//---------------------------------------------------------------------------------------------------------------
//
//  HAUD 2023.12.19
//
//  - XTS_TRANSPORT_LAYER
//
//  fb_Mover
//  - all positioning input is modulo value
//  - wrap MC function blocks
//
//
//---------------------------------------------------------------------------------------------------------------
// This SOFTWARE is provided as an Example by THE PROVIDER "as is" and "with all faults." THE PROVIDER makes no 
// representations or warranties of any kind concerning the safety, suitability, lack of viruses, inaccuracies, 
// typographical errors, or other harmful components of this SOFTWARE. There are inherent dangers in the use of 
// any software, and you are solely responsible for determining whether this SOFTWARE is compatible with your 
// equipment and other software installed on your equipment. You are also solely responsible for the protection 
// of your equipment and backup of your data, and THE PROVIDER will not be liable for any damages you may suffer 
// in connection with using, modifying, or distributing this SOFTWARE.
//---------------------------------------------------------------------------------------------------------------
FUNCTION_BLOCK fb_Mover IMPLEMENTS I_XtsTransport_Mover
VAR
  _nMoverId         : UINT;

  _sState           : STRING;

  _Master,
  _Mover            : REFERENCE TO AXIS_REF;
  _rLastPosition    : REFERENCE TO LREAL;
  _rLastGap         : REFERENCE TO LREAL;

  _RailLength       : LREAL;
  _nSyncStrategy    : Tc3_Mc3Definitions.MC_SYNC_STRATEGY := Tc3_Mc3Definitions.MC_SYNC_STRATEGY.mcSyncStrategySlow; // minimal movement with this strategy 

  // mover compact axis information
  _stInfo           : REFERENCE TO ST_MOVER_INFO; // ActPos, Enable, ...

  _bError           : BOOL;   // used in Cycle()
  _nErrorIdMover,             // used in Cycle()
  _nErrorIdPower    : UDINT;  // used in Cycle()

  //---------------------------------------------------------------------------
  // MC2 and CA function blocks
  //---------------------------------------------------------------------------
  _wMoverState      : DWORD;

  _fbMoveAbsCa      : Tc3_McCollisionAvoidance.MC_MoveAbsoluteCA;
  _fbSendAbsCa      : Tc3_McCollisionAvoidance.MC_MoveAbsoluteCA;
  _fbGearInPosCa    : Tc3_McCollisionAvoidance.MC_GearInPosCA;
  _fbHaltCa         : Tc3_McCollisionAvoidance.MC_HaltCA;

  _fbMoveAbs        : Tc2_MC2.MC_MoveAbsolute;
  _fbHalt           : Tc2_MC2.MC_Halt;
  _fbReset          : Tc2_MC2.MC_Reset;
  _fbStop           : Tc2_MC2.MC_Stop;

  _fbGearIn         : Tc2_MC2.MC_GearIn;
  _fbGearOut        : Tc2_MC2.MC_GearOut;

  _fbPower          : Tc2_MC2.MC_Power;

  _stMsg            : ST_Message;
  _eMessageLevel    : E_MessageType;
END_VAR

METHOD Check : BOOL
// check The thing that should not be

IF NOT (_nMoverId > 0)
THEN
  _sState                     := 'Mover: missing ID';
  RETURN;
END_IF

IF NOT __ISVALIDREF(_Mover)
THEN
  _sState                     := 'Mover: missing pointer';
  RETURN;
END_IF

IF NOT __ISVALIDREF(_rLastPosition)
THEN
  _sState                     := '_rLastPosition: missing pointer';
  RETURN;
END_IF

IF NOT __ISVALIDREF(_rLastGap)
THEN
  _sState                     := '_rLastGap: missing pointer';
  RETURN;
END_IF

IF NOT __ISVALIDREF(_stInfo)
THEN
  _sState                     := '_stInfo: missing pointer';
  RETURN;
END_IF

_sState                       := 'CHECK_DONE';
Check                         := TRUE;
END_METHOD

METHOD Cycle : E_PROGRESS
VAR_INST
  _eState             : E_PROGRESS;

  _rtrigMoverError,
  _rtrigPowerError    : Tc2_Standard.R_TRIG;
END_VAR
IF NOT Check() THEN Cycle := E_PROGRESS.PROGRESS_ERROR; RETURN; END_IF

_stMsg.eDevice            := e_Device.Mover + _nMoverId;

//-----------------------------------------------------------------------------------------------
// cyclic NC mapping
//-----------------------------------------------------------------------------------------------
_Mover();
//-----------------------------------------------------------------------------------------------


//-----------------------------------------------------------------------------------------------
// cyclic MC_Power
//-----------------------------------------------------------------------------------------------
_fbPower(
        Axis              := _Mover, 
        Enable_Positive   := TRUE, 
        Enable_Negative   := TRUE, 
        BufferMode        := MC_BufferMode.MC_Aborting);

_rtrigPowerError(CLK := _fbPower.Error);
_rtrigMoverError(CLK := _Mover.Status.Error); 

IF _rtrigMoverError.Q
THEN
  _bError                 := TRUE;  // deleted by Reset()
  // catch error
  _nErrorIdMover          := _Mover.Status.ErrorID;
  _stInfo.nErrorId        := _nErrorIdMover;

  _stMsg.eType            := E_MessageType.eMessageError;
  _stMsg.eSubdevice       := e_Subdevice.AxisControl;
  _stMsg.iErrorNumber     := _nErrorIdMover;
  _stMsg.sText            := 'Axis Error';
  f_MessageSet(_stMsg);
END_IF

IF _rtrigPowerError.Q
THEN
  _bError                 := TRUE;  // deleted by Reset()
  // catch error
  _nErrorIdPower          := _fbPower.ErrorID;
  _stInfo.nErrorId        := _nErrorIdPower;

  _stMsg.eType            := E_MessageType.eMessageError;
  _stMsg.eSubdevice       := e_Subdevice.AxisControl;
  _stMsg.iErrorNumber     := _nErrorIdMover;
  _stMsg.sText            := 'Axis Error';
  f_MessageSet(_stMsg);
END_IF
//-----------------------------------------------------------------------------------------------

//-----------------------------------------------------------------------------------------------
// cyclic state
//-----------------------------------------------------------------------------------------------
IF NOT _Mover.Status.ControlLoopClosed
THEN
  _eState                       := E_PROGRESS.PROGRESS_INIT;
ELSE
  _eState                       := E_PROGRESS.PROGRESS_WORKING;
END_IF
 
IF _bError
THEN
  _eState                       := E_PROGRESS.PROGRESS_ERROR;
END_IF
//-----------------------------------------------------------------------------------------------


//-----------------------------------------------------------------------------
// cyclic Mover info data
// get collision avoiding information from cyclic interface
//-----------------------------------------------------------------------------------------------
memcpy(ADR(_wMoverState), ADR(_Mover.NcToPlc.StateDWord2), SIZEOF(_wMoverState));

_stInfo.bMoverEnabled           := _Mover.Status.ControlLoopClosed;
_stInfo.bMoverError             := _bError;
_stInfo.bMoverCoupled           := _Mover.Status.Coupled;
_stInfo.bMoverStandstill        := _Mover.Status.NotMoving;
_stInfo.bMoverAvoidingCollision := _wMoverState.0;

_stInfo.rModuloActPos           := TO_REAL(_Mover.NcToPlc.ModuloActPos);
_stInfo.rAbsActPos              := TO_REAL(_Mover.NcToPlc.ActPos);

_stInfo.rModuloTargetPos        := TO_REAL(Tc2_Math.LMOD(_rLastPosition, _RailLength));
_stInfo.rAbsTargetPos           := TO_REAL(_rLastPosition);

IF (_Mover.NcToPlc.ActPos < _rLastPosition + 0.05) AND
   (_Mover.NcToPlc.ActPos > _rLastPosition - 0.05)
THEN
  _stInfo.bMoverInTarget        := TRUE;
ELSE
  _stInfo.bMoverInTarget        := FALSE;
END_IF
//-----------------------------------------------------------------------------

Cycle                           := _eState;
END_METHOD

METHOD Disable : E_PROGRESS
VAR_INPUT
  Execute             : BOOL;
END_VAR
VAR_INST
  _nErrorId           : UDINT;
  _eState             : E_PROGRESS;
END_VAR
IF NOT Execute THEN _eState  := E_PROGRESS.PROGRESS_INIT; END_IF 
IF NOT Check() THEN Disable  := E_PROGRESS.PROGRESS_ERROR; RETURN; END_IF


CASE _eState
OF
  E_PROGRESS.PROGRESS_INIT:
    IF Execute
    THEN
      _nErrorId               := 0;
      _eState                 := E_PROGRESS.PROGRESS_BUSY;
    END_IF
END_CASE
//-----------------------------------------------------------------------------
//-----------------------------------------------------------------------------
CASE _eState
OF
  E_PROGRESS.PROGRESS_BUSY:
    _eState                   := E_PROGRESS.PROGRESS_PREPARE;
    _fbPower.Enable           := FALSE;
END_CASE
//-----------------------------------------------------------------------------
//-----------------------------------------------------------------------------
CASE _eState
OF
  E_PROGRESS.PROGRESS_PREPARE:
    IF (_fbPower.Error)
    THEN
      _eState                 := E_PROGRESS.PROGRESS_ERROR;
      _nErrorId               := _fbPower.ErrorId;

      _stMsg.eType            := E_MessageType.eMessageError;
      _stMsg.eSubdevice       := e_Subdevice.fbPower;
      _stMsg.iErrorNumber     := _nErrorId;
      _stMsg.sText            := concat('Axis Disable: ', TO_STRING(_eState));
      f_MessageSet(_stMsg);

    ELSIF NOT (_Mover.Status.ControlLoopClosed)
    THEN
      _eState                 := E_PROGRESS.PROGRESS_DONE;

      IF (_eMessageLevel > E_MessageType.eMessageError)
      THEN
        _stMsg.eType          := E_MessageType.eMessageInfo;
        _stMsg.eSubdevice     := e_Subdevice.fbPower;
        _stMsg.iErrorNumber   := 0;
        _stMsg.sText          := concat('Axis Disable: ', TO_STRING(_eState));
        f_MessageSet(_stMsg);
      END_IF
    END_IF
END_CASE
//-----------------------------------------------------------------------------
//-----------------------------------------------------------------------------

Disable                       := _eState;
END_METHOD

METHOD Enable : E_PROGRESS
VAR_INPUT
  Execute             : BOOL;
END_VAR
VAR_INST
  _nErrorId           : UDINT;
  _eState             : E_PROGRESS;
END_VAR
IF NOT Execute THEN _eState  := E_PROGRESS.PROGRESS_INIT; END_IF 
IF NOT Check() THEN Enable   := E_PROGRESS.PROGRESS_ERROR; RETURN; END_IF


CASE _eState
OF
  E_PROGRESS.PROGRESS_INIT:
    IF Execute
    THEN
      _nErrorId               := 0;
      _eState                 := E_PROGRESS.PROGRESS_BUSY;
    END_IF
END_CASE
//-----------------------------------------------------------------------------
//-----------------------------------------------------------------------------
CASE _eState
OF
  E_PROGRESS.PROGRESS_BUSY:
    _eState                   := E_PROGRESS.PROGRESS_PREPARE;
    _fbPower.Enable           := TRUE;
END_CASE
//-----------------------------------------------------------------------------
//-----------------------------------------------------------------------------
CASE _eState
OF
  E_PROGRESS.PROGRESS_PREPARE:
    IF (_fbPower.Error)
    THEN
      _eState                 := E_PROGRESS.PROGRESS_ERROR;
      _nErrorId               := _fbPower.ErrorId;
      _stInfo.nErrorId        := _nErrorId;

      _stMsg.eType            := E_MessageType.eMessageError;
      _stMsg.eSubdevice       := e_Subdevice.fbPower;
      _stMsg.iErrorNumber     := _nErrorId;
      _stMsg.sText            := concat('Axis Enable: ', TO_STRING(_eState));
      f_MessageSet(_stMsg);

    ELSIF (_Mover.Status.ControlLoopClosed)
    THEN
      _eState                 := E_PROGRESS.PROGRESS_DONE;

      IF (_eMessageLevel > E_MessageType.eMessageError)
      THEN
        _stMsg.eType          := E_MessageType.eMessageInfo;
        _stMsg.eSubdevice     := e_Subdevice.fbPower;
        _stMsg.iErrorNumber   := _nErrorId;
        _stMsg.sText          := concat('Axis Enable: ', TO_STRING(_eState));
        f_MessageSet(_stMsg);
      END_IF
    END_IF
END_CASE
//-----------------------------------------------------------------------------
//-----------------------------------------------------------------------------

Enable                   := _eState;
END_METHOD

METHOD GearIn : E_PROGRESS;
VAR_INPUT
  Execute             : BOOL;
  stMoveData          : ST_MOVE_DATA;
  stGearData          : ST_GEAR_DATA;
END_VAR
VAR_INST
  _nErrorId           : UDINT;
  _eState             : E_PROGRESS;
END_VAR
IF NOT Execute THEN _eState  := E_PROGRESS.PROGRESS_INIT; END_IF 
IF NOT Check() THEN GearIn   := E_PROGRESS.PROGRESS_ERROR; RETURN; END_IF


CASE _eState
OF
  E_PROGRESS.PROGRESS_INIT:
    IF Execute
    THEN
      _nErrorId               := 0;
      _eState                 := E_PROGRESS.PROGRESS_BUSY;

      IF NOT __ISVALIDREF(_Master)
      THEN
        _bError               := TRUE;
        _nErrorId             := 666;
        _eState               := E_PROGRESS.PROGRESS_ERROR;

        _stMsg.eType          := E_MessageType.eMessageError;
        _stMsg.eSubdevice     := e_Subdevice.fbGearIn;
        _stMsg.iErrorNumber   := _nErrorId;
        _stMsg.sText          := concat('Invalid Master Ref: ', TO_STRING(_eState));
        f_MessageSet(_stMsg);
      END_IF
    END_IF
END_CASE
//-----------------------------------------------------------------------------
//-----------------------------------------------------------------------------
CASE _eState
OF
  E_PROGRESS.PROGRESS_BUSY:
    _eState                   := E_PROGRESS.PROGRESS_PREPARE;
    _fbPower.Override         := stMoveData.rOverride;

    _fbGearIn(
            Master            := _Master, 
            Slave             := _Mover,
            Execute           := FALSE,
            RatioNumerator    := stGearData.rGearNumerator,
            RatioDenominator  := stGearData.iGearDenumerator, 
            Acceleration      := stMoveData.rAcc, 
            Deceleration      := stMoveData.rAcc, 
            Jerk              := stMoveData.rJerk, 
            BufferMode        := Tc2_MC2.MC_BufferMode.MC_Aborting);
END_CASE
//-----------------------------------------------------------------------------
//-----------------------------------------------------------------------------
CASE _eState
OF
  E_PROGRESS.PROGRESS_PREPARE:
    _fbGearIn(
            Master            := _Master, 
            Slave             := _Mover,
            Execute           := TRUE);

    IF _fbGearIn.Error
    THEN
      _bError                 := TRUE;
      _nErrorId               := _fbGearIn.ErrorID;
      _eState                 := E_PROGRESS.PROGRESS_ERROR;

      _stMsg.eType            := E_MessageType.eMessageError;
      _stMsg.eSubdevice       := e_Subdevice.fbGearIn;
      _stMsg.iErrorNumber     := _nErrorId;
      _stMsg.sText            := TO_STRING(_eState);
      f_MessageSet(_stMsg);

    ELSIF _fbGearIn.InGear
    THEN
      _eState                 := E_PROGRESS.PROGRESS_DONE;

      IF (_eMessageLevel > E_MessageType.eMessageError)
      THEN
        _stMsg.eType          := E_MessageType.eMessageInfo;
        _stMsg.eSubdevice     := e_Subdevice.fbGearIn;
        _stMsg.iErrorNumber   := _nErrorId;
        _stMsg.sText          := TO_STRING(_eState);
        f_MessageSet(_stMsg);
      END_IF
    END_IF
END_CASE
//-----------------------------------------------------------------------------
//-----------------------------------------------------------------------------
CASE _eState
OF
  E_PROGRESS.PROGRESS_ERROR,
  E_PROGRESS.PROGRESS_DONE:
    _stInfo.nErrorId          := _nErrorId;
    _fbGearIn(
            Master            := _Master, 
            Slave             := _Mover,
            Execute           := FALSE);
END_CASE
//-----------------------------------------------------------------------------
//-----------------------------------------------------------------------------

GearIn                        := _eState;
END_METHOD

METHOD GearInPosCa : E_PROGRESS
VAR_INPUT
  Execute             : BOOL;
  stMoveData          : ST_MOVE_DATA;
  stGearData          : ST_GEAR_DATA;  
END_VAR
VAR_INST
  _nErrorId           : UDINT;
  _rPosLate,
  _rPos               : LREAL;
  _eState             : E_PROGRESS;

  _rModActPos         : LREAL;
END_VAR
IF NOT Execute THEN _eState       := E_PROGRESS.PROGRESS_INIT; END_IF 
IF NOT Check() THEN GearInPosCa   := E_PROGRESS.PROGRESS_ERROR; RETURN; END_IF


CASE _eState
OF
  E_PROGRESS.PROGRESS_INIT:
    IF Execute
    THEN
      _rPosLate               := 0.0;
      _nErrorId               := 0;
      _eState                 := E_PROGRESS.PROGRESS_BUSY;
      _rModActPos             := Tc2_Math.LMOD(_Mover.NcToPlc.SetPos, _RailLength);

      IF NOT __ISVALIDREF(_Master)
      THEN
        _bError               := TRUE;
        _nErrorId             := 666;
        _eState               := E_PROGRESS.PROGRESS_ERROR;

        _stMsg.eType          := E_MessageType.eMessageError;
        _stMsg.eSubdevice     := e_Subdevice.fbGearInPosCa;
        _stMsg.iErrorNumber   := _nErrorId;
        _stMsg.sText          := concat('Invalid Master Ref: ', TO_STRING(_eState));
        f_MessageSet(_stMsg);

      ELSIF (_rModActPos > stGearData.rModuloSyncPosSlave + stMoveData.rDelta)
      THEN
        _bError               := TRUE;
        _rPosLate             := _rModActPos;
        _rPos                 := stGearData.rModuloSyncPosSlave + stMoveData.rDelta;

        _nErrorId             := 667;
        _eState               := E_PROGRESS.PROGRESS_ERROR;

        _stMsg.eType          := E_MessageType.eMessageError;
        _stMsg.eSubdevice     := e_Subdevice.fbGearInPosCa;
        _stMsg.iErrorNumber   := _nErrorId;
        _stMsg.sText          := concat('_rModActPos: ', TO_STRING(_rPosLate));
        _stMsg.sText          := concat(_stMsg.sText, '; ModuloSyncPosSlave + stMoveData.Delta: ');
        _stMsg.sText          := concat(_stMsg.sText, TO_STRING(_rPos));
        f_MessageSet(_stMsg);
      END_IF
    END_IF
END_CASE
//-----------------------------------------------------------------------------
//-----------------------------------------------------------------------------
CASE _eState
OF
  E_PROGRESS.PROGRESS_BUSY:
    _eState                   := E_PROGRESS.PROGRESS_PREPARE;

    _fbPower.Override         := stMoveData.rOverride;

    _fbGearInPosCa(
        Master                := _Master, 
        Slave                 := _Mover, 
        Execute               := FALSE, 
        ContinuousUpdate      := TRUE, 
        RatioNumerator        := stGearData.rGearNumerator, 
        RatioDenumerator      := stGearData.iGearDenumerator, 

        MasterSyncPosition    := _Master.NcToPlc.ActPos 
                               + stGearData.rDeltaToMasterPos,                            // absolute position

        SlaveSyncPosition     := ABS(_Mover.NcToPlc.ModuloActTurns)*_RailLength
                               + stGearData.rModuloSyncPosSlave,                          // absolute position

        SyncStrategy          := _nSyncStrategy,  
        SyncMode              := Tc3_Mc3Definitions.MC_SYNC_MODE.mcSyncModeNonModulo,     // all positions as absolute value
        MasterStartDistance   := stGearData.rMasterStartDistance,                         // if <> 0 --> master has to move before this fb does anything
        Velocity              := stMoveData.rVelo, 
        Acceleration          := stMoveData.rAcc, 
        Deceleration          := stMoveData.rAcc, 
        Jerk                  := stMoveData.rJerk, 
        Gap                   := stMoveData.rGap, 
        BufferMode            := Tc3_Mc3Definitions.MC_BUFFER_MODE.mcAborting);

        IF (_eMessageLevel > E_MessageType.eMessageInfo)
        THEN
          _stMsg.eType        := E_MessageType.eMessageVerbose;
          _stMsg.eSubdevice   := e_Subdevice.fbGearInPosCa;
          _stMsg.iErrorNumber := _nErrorId;
          _stMsg.sText        := TO_STRING(_eState);
          f_MessageSet(_stMsg);
        END_IF
END_CASE
//-----------------------------------------------------------------------------
//-----------------------------------------------------------------------------
CASE _eState
OF
  E_PROGRESS.PROGRESS_PREPARE:
    _fbGearInPosCa(
        Master                := _Master, 
        Slave                 := _Mover, 
        Execute               := TRUE, 
        ContinuousUpdate      := TRUE);

    IF _fbGearInPosCa.Error
    THEN
      _bError                 := TRUE;
      _nErrorId               := _fbGearInPosCa.ErrorId;
      _stInfo.nErrorId        := _nErrorId;
      _fbGearInPosCa(
        Master                := _Master, 
        Slave                 := _Mover, 
        Execute               := FALSE, 
        ContinuousUpdate      := TRUE);

      _eState                 := E_PROGRESS.PROGRESS_ERROR;

      _stMsg.eType          := E_MessageType.eMessageError;
      _stMsg.eSubdevice     := e_Subdevice.fbGearInPosCa;
      _stMsg.iErrorNumber   := _nErrorId;
      _stMsg.sText          := TO_STRING(_eState);
      f_MessageSet(_stMsg);

    ELSIF _fbGearInPosCa.CommandAborted
    THEN
      _bError                 := TRUE;
      _eState                 := E_PROGRESS.PROGRESS_OCCUPIED;

      _stMsg.eType            := E_MessageType.eMessageWarning;
      _stMsg.eSubdevice       := e_Subdevice.fbGearInPosCa;
      _stMsg.iErrorNumber     := _nErrorId;
      _stMsg.sText            := TO_STRING(_eState);
      f_MessageSet(_stMsg);

    ELSIF _fbGearInPosCa.InSync
    THEN
      _eState                 := E_PROGRESS.PROGRESS_DONE;

      IF (_eMessageLevel > E_MessageType.eMessageError)
      THEN
        _stMsg.eType          := E_MessageType.eMessageInfo;
        _stMsg.eSubdevice     := e_Subdevice.fbGearInPosCa;
        _stMsg.iErrorNumber   := _nErrorId;
        _stMsg.sText          := TO_STRING(_eState);
        f_MessageSet(_stMsg);
      END_IF
      _fbGearInPosCa(
        Master                := _Master, 
        Slave                 := _Mover, 
        Execute               := FALSE, 
        ContinuousUpdate      := TRUE);
    END_IF
END_CASE
//-----------------------------------------------------------------------------
//-----------------------------------------------------------------------------

GearInPosCa                   := _eState;
END_METHOD

METHOD GearOut : E_PROGRESS
VAR_INPUT
  Execute             : BOOL;
END_VAR
VAR_INST
  _nErrorId           : UDINT;
  _eState             : E_PROGRESS;
END_VAR
IF NOT Execute THEN _eState  := E_PROGRESS.PROGRESS_INIT; END_IF 
IF NOT Check() THEN GearOut  := E_PROGRESS.PROGRESS_ERROR; RETURN; END_IF


CASE _eState
OF
  E_PROGRESS.PROGRESS_INIT:
    IF Execute
    THEN
      _nErrorId               := 0;
      _eState                 := E_PROGRESS.PROGRESS_BUSY;
    END_IF
END_CASE
//-----------------------------------------------------------------------------
//-----------------------------------------------------------------------------
CASE _eState
OF
  E_PROGRESS.PROGRESS_BUSY:
    _eState                   := E_PROGRESS.PROGRESS_PREPARE;
    _fbGearOut(
            Slave             := _Mover, 
            Execute           := FALSE);

    IF (_eMessageLevel > E_MessageType.eMessageError)
    THEN
      _stMsg.eType            := E_MessageType.eMessageInfo;
      _stMsg.eSubdevice       := e_Subdevice.fbGearOut;
      _stMsg.iErrorNumber     := _nErrorId;
      _stMsg.sText            := TO_STRING(_eState);
      f_MessageSet(_stMsg);
    END_IF
END_CASE
//-----------------------------------------------------------------------------
//-----------------------------------------------------------------------------
CASE _eState
OF
  E_PROGRESS.PROGRESS_PREPARE:
    _fbGearOut(
            Slave             := _Mover, 
            Execute           := TRUE);

    IF _fbGearOut.Error
    THEN
      _bError                 := TRUE;
      _nErrorId               := _fbGearOut.ErrorID;
      _eState                 := E_PROGRESS.PROGRESS_ERROR;

      _stMsg.eType            := E_MessageType.eMessageError;
      _stMsg.eSubdevice       := e_Subdevice.fbGearOut;
      _stMsg.iErrorNumber     := _nErrorId;
      _stMsg.sText            := TO_STRING(_eState);
      f_MessageSet(_stMsg);

    ELSIF (_Mover.NcToPlc.CoupleState = 0)
    THEN
      _eState                 := E_PROGRESS.PROGRESS_DONE;

      IF (_eMessageLevel > E_MessageType.eMessageError)
      THEN
        _stMsg.eType          := E_MessageType.eMessageInfo;
        _stMsg.eSubdevice     := e_Subdevice.fbGearOut;
        _stMsg.iErrorNumber   := _nErrorId;
        _stMsg.sText          := TO_STRING(_eState);
        f_MessageSet(_stMsg);
      END_IF
    END_IF
END_CASE
//-----------------------------------------------------------------------------
//-----------------------------------------------------------------------------
CASE _eState
OF
  E_PROGRESS.PROGRESS_ERROR,
  E_PROGRESS.PROGRESS_DONE:
    _stInfo.nErrorId          := _nErrorId;
    _fbGearOut(
            Slave             := _Mover, 
            Execute           := FALSE);
END_CASE
//-----------------------------------------------------------------------------
//-----------------------------------------------------------------------------

GearOut                       := _eState;
END_METHOD

METHOD Halt : E_PROGRESS
VAR_INPUT
  Execute             : BOOL;
  stMoveData          : ST_MOVE_DATA;
END_VAR
VAR_INST
  _nErrorId           : UDINT;
  _eState             : E_PROGRESS;
END_VAR
IF NOT Execute 
THEN 
	_eState := E_PROGRESS.PROGRESS_INIT; 
END_IF 
IF NOT Check() 
THEN 
	Halt := E_PROGRESS.PROGRESS_ERROR; 
	RETURN; 
END_IF


CASE _eState
OF
  E_PROGRESS.PROGRESS_INIT:
    IF Execute
    THEN
      _nErrorId               := 0;
      _eState                 := E_PROGRESS.PROGRESS_BUSY;
    END_IF
END_CASE
//-----------------------------------------------------------------------------
//-----------------------------------------------------------------------------
CASE _eState
OF
  E_PROGRESS.PROGRESS_BUSY:
    _eState                   := E_PROGRESS.PROGRESS_PREPARE;
    _fbHalt(
            Axis              := _Mover, 
            Execute           := FALSE, 
            Deceleration      := stMoveData.rAcc, 
            Jerk              := stMoveData.rJerk, 
            BufferMode        := Tc2_MC2.MC_BufferMode.MC_Aborting);

    IF (_eMessageLevel > E_MessageType.eMessageInfo)
    THEN
      _stMsg.eType            := E_MessageType.eMessageVerbose;
      _stMsg.eSubdevice       := e_Subdevice.fbHalt;
      _stMsg.iErrorNumber     := _nErrorId;
      _stMsg.sText            := TO_STRING(_eState);
      f_MessageSet(_stMsg);
    END_IF
END_CASE
//-----------------------------------------------------------------------------
//-----------------------------------------------------------------------------
CASE _eState
OF
  E_PROGRESS.PROGRESS_PREPARE:
    _fbHalt(Axis              := _Mover, 
            Execute           := TRUE, 
            Deceleration      := stMoveData.rAcc, 
            Jerk              := stMoveData.rJerk, 
            BufferMode        := Tc2_MC2.MC_BufferMode.MC_Aborting);

    IF _fbHalt.Error
    THEN
      _bError                 := TRUE;
      _nErrorId               := _fbHalt.ErrorID;
      _eState                 := E_PROGRESS.PROGRESS_ERROR;

      _stMsg.eType            := E_MessageType.eMessageError;
      _stMsg.eSubdevice       := e_Subdevice.fbHalt;
      _stMsg.iErrorNumber     := _nErrorId;
      _stMsg.sText            := TO_STRING(_eState);
      f_MessageSet(_stMsg);

    ELSIF NOT _Mover.Status.Moving
    THEN
      _eState                 := E_PROGRESS.PROGRESS_DONE;

      IF (_eMessageLevel > E_MessageType.eMessageError)
      THEN
        _stMsg.eType          := E_MessageType.eMessageInfo;
        _stMsg.eSubdevice     := e_Subdevice.fbHalt;
        _stMsg.iErrorNumber   := _nErrorId;
        _stMsg.sText          := TO_STRING(_eState);
        f_MessageSet(_stMsg);
      END_IF
    END_IF
END_CASE
//-----------------------------------------------------------------------------
//-----------------------------------------------------------------------------
CASE _eState
OF
  E_PROGRESS.PROGRESS_ERROR,
  E_PROGRESS.PROGRESS_DONE:
    _stInfo.nErrorId          := _nErrorId;
    _fbHalt(
            Axis              := _Mover, 
            Execute           := FALSE);
END_CASE
//-----------------------------------------------------------------------------
//-----------------------------------------------------------------------------

Halt                          := _eState;
END_METHOD

METHOD HaltCa : E_PROGRESS
VAR_INPUT
  Execute             : BOOL;
  stMoveData          : ST_MOVE_DATA;
END_VAR
VAR_INST
  _nErrorId           : UDINT;
  _eState             : E_PROGRESS;
END_VAR
IF NOT Execute 
THEN 
	_eState := E_PROGRESS.PROGRESS_INIT; 
END_IF 
IF NOT Check() 
THEN 
	HaltCa := E_PROGRESS.PROGRESS_ERROR; 
	RETURN; 
END_IF


CASE _eState
OF
  E_PROGRESS.PROGRESS_INIT:
    IF Execute
    THEN
      _nErrorId               := 0;
      _eState                 := E_PROGRESS.PROGRESS_BUSY;
    END_IF
END_CASE
//-----------------------------------------------------------------------------
//-----------------------------------------------------------------------------
CASE _eState
OF
  E_PROGRESS.PROGRESS_BUSY:
    _eState                   := E_PROGRESS.PROGRESS_PREPARE;
    _fbHaltCa(
            Axis              := _Mover, 
            Execute           := FALSE, 
            Deceleration      := stMoveData.rAcc, 
            Jerk              := stMoveData.rJerk, 
            Gap               := stMoveData.rGap);

    IF (_eMessageLevel > E_MessageType.eMessageInfo)
    THEN
      _stMsg.eType            := E_MessageType.eMessageVerbose;
      _stMsg.eSubdevice       := e_Subdevice.fbHaltCa;
      _stMsg.iErrorNumber     := _nErrorId;
      _stMsg.sText            := TO_STRING(_eState);
      f_MessageSet(_stMsg);
    END_IF
END_CASE
//-----------------------------------------------------------------------------
//-----------------------------------------------------------------------------
CASE _eState
OF
  E_PROGRESS.PROGRESS_PREPARE:
    _fbHaltCa(
            Axis              := _Mover, 
            Execute           := TRUE, 
            Deceleration      := stMoveData.rAcc, 
            Jerk              := stMoveData.rJerk, 
            Gap               := stMoveData.rGap);

    IF _fbHaltCa.Error
    THEN
      _bError                 := TRUE;
      _nErrorId               := _fbHalt.ErrorID;
      _eState                 := E_PROGRESS.PROGRESS_ERROR;

      _stMsg.eType            := E_MessageType.eMessageError;
      _stMsg.eSubdevice       := e_Subdevice.fbHaltCa;
      _stMsg.iErrorNumber     := _nErrorId;
      _stMsg.sText            := TO_STRING(_eState);
      f_MessageSet(_stMsg);

    ELSIF NOT _Mover.Status.Moving
    THEN
      _eState                 := E_PROGRESS.PROGRESS_DONE;

      IF (_eMessageLevel > E_MessageType.eMessageError)
      THEN
        _stMsg.eType          := E_MessageType.eMessageInfo;
        _stMsg.eSubdevice     := e_Subdevice.fbHaltCa;
        _stMsg.iErrorNumber   := _nErrorId;
        _stMsg.sText          := TO_STRING(_eState);
        f_MessageSet(_stMsg);
      END_IF
    END_IF
END_CASE
//-----------------------------------------------------------------------------
//-----------------------------------------------------------------------------
CASE _eState
OF
  E_PROGRESS.PROGRESS_ERROR,
  E_PROGRESS.PROGRESS_DONE:
    _stInfo.nErrorId          := _nErrorId;
    _fbHaltCa(
            Axis              := _Mover, 
            Execute           := FALSE);
END_CASE
//-----------------------------------------------------------------------------
//-----------------------------------------------------------------------------

HaltCa                          := _eState;
END_METHOD

PROPERTY LastGap : REFERENCE to lreal
SET
_rLastGap REF= LastGap;
END_SET
END_PROPERTY

PROPERTY LastPosition : REFERENCE to LREAL
SET
_rLastPosition REF= LastPosition;
END_SET
END_PROPERTY

PROPERTY Master : REFERENCE to AXIS_REF
SET
_Master REF= Master;
END_SET
END_PROPERTY

PROPERTY MessageLevel : e_messagetype
SET
_eMessageLevel := MessageLevel;
END_SET
END_PROPERTY

PROPERTY ModuloTurn : dint
GET
ModuloTurn := _Mover.NcToPlc.ModuloSetTurns;
END_GET
END_PROPERTY

PROPERTY Mover : REFERENCE to AXIS_REF
SET
_Mover REF= Mover;
END_SET
END_PROPERTY

PROPERTY MoverId : uint
SET
_nMoverId := MoverId;
END_SET
END_PROPERTY

PROPERTY MoverInfo : REFERENCE to ST_MOVER_INFO
SET


	_stInfo ref= MoverInfo;
END_SET
END_PROPERTY

METHOD MoveToPos : E_PROGRESS
VAR_INPUT
  Execute             : BOOL;
  stMoveData          : ST_MOVE_DATA;
END_VAR
VAR_INST
  _nErrorId           : UDINT;
  _rDelta,
  _rPos               : LREAL;
  _eState             : E_PROGRESS;
END_VAR
IF NOT Execute THEN _eState  := E_PROGRESS.PROGRESS_INIT; END_IF 
IF NOT Check() THEN MoveToPos   := E_PROGRESS.PROGRESS_ERROR; RETURN; END_IF


CASE _eState
OF
  E_PROGRESS.PROGRESS_INIT:
    IF Execute
    THEN
      _nErrorId               := 0;
      _rDelta                 := SEL((stMoveData.rDelta < 0.01), stMoveData.rDelta, 0.05);
      _eState                 := E_PROGRESS.PROGRESS_BUSY;
    END_IF
END_CASE
//-----------------------------------------------------------------------------
//-----------------------------------------------------------------------------
CASE _eState
OF
  E_PROGRESS.PROGRESS_BUSY:
    _eState                   := E_PROGRESS.PROGRESS_PREPARE;
    _fbPower.Override         := stMoveData.rOverride;

    _rPos                     := ABS(_Mover.NcToPlc.ModuloActTurns)* _RailLength + stMoveData.rPos;


    _rLastPosition            := _rPos;
    //_rLastGap                 := stMoveData.rGap;

    _fbMoveAbs(
            Axis              := _Mover, 
            Execute           := FALSE, 
            Position          := _rPos, 
            Velocity          := stMoveData.rVelo, 
            Acceleration      := stMoveData.rAcc, 
            Deceleration      := stMoveData.rAcc, 
            Jerk              := stMoveData.rJerk, 
            BufferMode        := Tc2_MC2.MC_BufferMode.MC_Aborting);

      IF (_eMessageLevel > E_MessageType.eMessageInfo)
      THEN
        _stMsg.eType          := E_MessageType.eMessageVerbose;
        _stMsg.eSubdevice     := e_Subdevice.fbMovePtP;
        _stMsg.iErrorNumber   := _nErrorId;
        _stMsg.sText          := concat(TO_STRING(_eState), ': ');
        _stMsg.sText          := concat(_stMsg.sText, concat('stMoveData.rPos: ', TO_STRING(stMoveData.rPos)));
        f_MessageSet(_stMsg);
      END_IF
END_CASE
//-----------------------------------------------------------------------------
//-----------------------------------------------------------------------------
CASE _eState
OF
  E_PROGRESS.PROGRESS_PREPARE:
    _fbMoveAbs(
            Axis              := _Mover, 
            Execute           := TRUE, 
            Position          := _rPos, 
            Velocity          := stMoveData.rVelo, 
            Acceleration      := stMoveData.rAcc, 
            Deceleration      := stMoveData.rAcc, 
            Jerk              := stMoveData.rJerk, 
            BufferMode        := Tc2_MC2.MC_BufferMode.MC_Aborting);

    IF _fbMoveAbs.Error
    THEN
      _bError                 := TRUE;
      _nErrorId               := _fbMoveAbs.ErrorId;
      _eState                 := E_PROGRESS.PROGRESS_ERROR;

      _stMsg.eType            := E_MessageType.eMessageError;
      _stMsg.eSubdevice       := e_Subdevice.fbMovePtP;
      _stMsg.iErrorNumber     := _nErrorId;
      _stMsg.sText            := TO_STRING(_eState);
      f_MessageSet(_stMsg);

    ELSIF _fbMoveAbs.Active OR 
          _fbMoveAbs.Done
		THEN
      _eState                 := E_PROGRESS.PROGRESS_WORKING;

      IF (_eMessageLevel = E_MessageType.eMessageVerbose)
      THEN
        _stMsg.eType          := E_MessageType.eMessageVerbose;
        _stMsg.eSubdevice     := e_Subdevice.fbMovePtP;
        _stMsg.iErrorNumber   := _nErrorId;
        _stMsg.sText          := concat(TO_STRING(_eState), ': ');
        _stMsg.sText          := concat(_stMsg.sText, '.ModuloActPos: ');
        _stMsg.sText          := concat(_stMsg.sText, TO_STRING(_Mover.NcToPlc.ModuloActPos));
        f_MessageSet(_stMsg);
      END_IF
    END_IF
END_CASE
//-----------------------------------------------------------------------------
//-----------------------------------------------------------------------------
CASE _eState
OF
  E_PROGRESS.PROGRESS_WORKING:
    _fbMoveAbs(
          Axis                := _Mover);

    IF _fbMoveAbs.Error
    THEN
      _bError                 := TRUE;
      _nErrorId               := _fbMoveAbs.ErrorId;
      _stInfo.nErrorId        := _nErrorId;
      _eState                 := E_PROGRESS.PROGRESS_ERROR;

      _stMsg.eType            := E_MessageType.eMessageError;
      _stMsg.eSubdevice       := e_Subdevice.fbMovePtP;
      _stMsg.iErrorNumber     := _nErrorId;
      _stMsg.sText            := TO_STRING(_eState);
      f_MessageSet(_stMsg);

      _fbMoveAbs( 
            Axis              := _Mover, 
            Execute           := FALSE);


    ELSIF (_Mover.NcToPlc.ActPos > _fbMoveAbs.Position - _rDelta) AND
          (_Mover.NcToPlc.ActPos < _fbMoveAbs.Position + _rDelta)
    THEN
      IF NOT _Mover.Status.Moving
      THEN
        _eState               := E_PROGRESS.PROGRESS_DONE;

        IF (_eMessageLevel > E_MessageType.eMessageError)
        THEN
          _stMsg.eType        := E_MessageType.eMessageInfo;
          _stMsg.eSubdevice   := e_Subdevice.fbMovePtP;
          _stMsg.iErrorNumber := _nErrorId;
          _stMsg.sText        := concat(TO_STRING(_eState), ': ');
          _stMsg.sText        := concat(_stMsg.sText, concat('ModActPos: ', TO_STRING(_Mover.NcToPlc.ModuloActPos)));
          f_MessageSet(_stMsg);
        END_IF
      _fbMoveAbs( 
            Axis              := _Mover, 
            Execute           := FALSE);
      END_IF
    END_IF
END_CASE
//-----------------------------------------------------------------------------
//-----------------------------------------------------------------------------

MoveToPos                   := _eState;
END_METHOD

METHOD MoveToPosCa : E_PROGRESS
VAR_INPUT
  Execute             : BOOL;
  stMoveData          : ST_MOVE_DATA;
END_VAR
VAR_INST
  _nErrorId           : UDINT;
  _rDelta,
  _rPos               : LREAL;
  _eState             : E_PROGRESS;
END_VAR
IF NOT Execute THEN _eState  := E_PROGRESS.PROGRESS_INIT; END_IF 
IF NOT Check() THEN MoveToPosCa   := E_PROGRESS.PROGRESS_ERROR; RETURN; END_IF


CASE _eState
OF
  E_PROGRESS.PROGRESS_INIT:
    IF Execute
    THEN
      _nErrorId               := 0;
      _rDelta                 := SEL((stMoveData.rDelta < 0.01), stMoveData.rDelta, 0.05);
      _eState                 := E_PROGRESS.PROGRESS_BUSY;
    END_IF
END_CASE
//-----------------------------------------------------------------------------
//-----------------------------------------------------------------------------
CASE _eState
OF
  E_PROGRESS.PROGRESS_BUSY:
    _eState                   := E_PROGRESS.PROGRESS_PREPARE;
    _fbPower.Override         := stMoveData.rOverride;

    _rPos                     := ABS(_Mover.NcToPlc.ModuloActTurns)* _RailLength + stMoveData.rPos;


    _rLastPosition            := _rPos;
    _rLastGap                 := stMoveData.rGap;

    _fbMoveAbsCa( 
            Axis              := _Mover, 
            Execute           := FALSE, 
            ContinuousUpdate  := TRUE, 
            Position          := _rPos,
            Velocity          := stMoveData.rVelo, 
            Acceleration      := stMoveData.rAcc, 
            Deceleration      := stMoveData.rAcc, 
            Jerk              := stMoveData.rJerk, 
            Gap               := stMoveData.rGap, 
            BufferMode        := Tc3_Mc3Definitions.MC_BUFFER_MODE.mcAborting);

    IF (_eMessageLevel > E_MessageType.eMessageInfo)
    THEN
      _stMsg.eType            := E_MessageType.eMessageVerbose;
      _stMsg.eSubdevice       := e_Subdevice.fbMoveToPosCa;
      _stMsg.iErrorNumber     := _nErrorId;
      _stMsg.sText            := concat(TO_STRING(_eState), ': ');
      _stMsg.sText            := concat(_stMsg.sText, concat('stMoveData.rPos: ', TO_STRING(stMoveData.rPos)));
      f_MessageSet(_stMsg);
    END_IF
END_CASE
//-----------------------------------------------------------------------------
//-----------------------------------------------------------------------------
CASE _eState
OF
  E_PROGRESS.PROGRESS_PREPARE:
    _fbMoveAbsCa( 
            Axis              := _Mover, 
            Execute           := TRUE, 
            ContinuousUpdate  := TRUE, 
            Position          := _rPos,
            Velocity          := stMoveData.rVelo, 
            Acceleration      := stMoveData.rAcc, 
            Deceleration      := stMoveData.rAcc, 
            Jerk              := stMoveData.rJerk, 
            Gap               := stMoveData.rGap, 
            BufferMode        := Tc3_Mc3Definitions.MC_BUFFER_MODE.mcAborting);

    IF _fbMoveAbsCa.Error
    THEN
      _bError                 := TRUE;
      _nErrorId               := _fbMoveAbsCa.ErrorId;
      _stInfo.nErrorId        := _nErrorId;
      _eState                 := E_PROGRESS.PROGRESS_ERROR;

      _stMsg.eType            := E_MessageType.eMessageError;
      _stMsg.eSubdevice       := e_Subdevice.fbMoveToPosCa;
      _stMsg.iErrorNumber     := _nErrorId;
      _stMsg.sText            := TO_STRING(_eState);
      f_MessageSet(_stMsg);

    ELSIF _fbMoveAbsCa.Active OR 
          _fbMoveAbsCa.Done
		THEN
      _eState                 := E_PROGRESS.PROGRESS_WORKING;

      IF (_eMessageLevel = E_MessageType.eMessageVerbose)
      THEN
        _stMsg.eType          := E_MessageType.eMessageVerbose;
        _stMsg.eSubdevice     := e_Subdevice.fbMoveToPosCa;
        _stMsg.iErrorNumber   := _nErrorId;
        _stMsg.sText          := concat(TO_STRING(_eState), ': ');
        _stMsg.sText          := concat(_stMsg.sText, '.ModuloActPos: ');
        _stMsg.sText          := concat(_stMsg.sText, TO_STRING(_Mover.NcToPlc.ModuloActPos));
        f_MessageSet(_stMsg);
      END_IF
    END_IF
END_CASE
//-----------------------------------------------------------------------------
//-----------------------------------------------------------------------------
CASE _eState
OF
  E_PROGRESS.PROGRESS_WORKING:
    _fbMoveAbsCa(
          Axis                := _Mover);

    IF _fbMoveAbsCa.Error
    THEN
      _bError                 := TRUE;
      _nErrorId               := _fbMoveAbsCa.ErrorId;
      _stInfo.nErrorId        := _nErrorId;
      _fbMoveAbsCa( 
            Axis              := _Mover, 
            Execute           := FALSE);

      _eState                 := E_PROGRESS.PROGRESS_ERROR;

      _stMsg.eType            := E_MessageType.eMessageError;
      _stMsg.eSubdevice       := e_Subdevice.fbMoveToPosCa;
      _stMsg.iErrorNumber     := _nErrorId;
      _stMsg.sText            := concat(TO_STRING(_eState), ': ');
      _stMsg.sText            := concat(_stMsg.sText, concat('ModActPos: ', TO_STRING(_Mover.NcToPlc.ModuloActPos)));

      f_MessageSet(_stMsg);

    ELSIF (_Mover.NcToPlc.ActPos > _fbMoveAbsCa.Position - _rDelta) AND
          (_Mover.NcToPlc.ActPos < _fbMoveAbsCa.Position + _rDelta)
    THEN
      IF NOT _Mover.Status.Moving
      THEN
        _eState               := E_PROGRESS.PROGRESS_DONE;

        IF (_eMessageLevel > E_MessageType.eMessageError)
        THEN
          _stMsg.eType        := E_MessageType.eMessageInfo;
          _stMsg.eSubdevice   := e_Subdevice.fbMoveToPosCa;
          _stMsg.iErrorNumber := _nErrorId;
          _stMsg.sText        := concat(TO_STRING(_eState), ': ');
          _stMsg.sText        := concat(_stMsg.sText, concat('ModActPos: ', TO_STRING(_Mover.NcToPlc.ModuloActPos)));
          f_MessageSet(_stMsg);
        END_IF
      _fbMoveAbsCa( 
            Axis              := _Mover, 
            Execute           := FALSE);
      END_IF
    END_IF
END_CASE
//-----------------------------------------------------------------------------
//-----------------------------------------------------------------------------

MoveToPosCa                   := _eState;
END_METHOD

PROPERTY RailLength : LREAL
GET
RailLength := _RailLength;
END_GET
SET
_RailLength := RailLength;
END_SET
END_PROPERTY

METHOD Reset : E_PROGRESS
VAR_INPUT
  Execute             : BOOL;
END_VAR
VAR_INST
  _nErrorId           : UDINT;
  _eState             : E_PROGRESS;
END_VAR
IF NOT Execute THEN _eState  := E_PROGRESS.PROGRESS_INIT; END_IF 
IF NOT Check() THEN Reset    := E_PROGRESS.PROGRESS_ERROR; RETURN; END_IF


CASE _eState
OF
  E_PROGRESS.PROGRESS_INIT:
    IF Execute
    THEN
      _stInfo.nErrorId        :=
      _nErrorId               := 0;
      _eState                 := E_PROGRESS.PROGRESS_BUSY;
    END_IF
END_CASE
//-----------------------------------------------------------------------------
//-----------------------------------------------------------------------------
CASE _eState
OF
  E_PROGRESS.PROGRESS_BUSY:
    _eState                   := E_PROGRESS.PROGRESS_PREPARE;
    _fbReset(
            Axis              := _Mover, 
            Execute           := FALSE);

    IF (_eMessageLevel > E_MessageType.eMessageInfo)
    THEN
      _stMsg.eType            := E_MessageType.eMessageVerbose;
      _stMsg.eSubdevice       := e_Subdevice.fbReset;
      _stMsg.iErrorNumber     := _nErrorId;
      _stMsg.sText            := TO_STRING(_eState);
      f_MessageSet(_stMsg);
    END_IF
END_CASE
//-----------------------------------------------------------------------------
//-----------------------------------------------------------------------------
CASE _eState
OF
  E_PROGRESS.PROGRESS_PREPARE:
    _fbReset(
            Axis              := _Mover, 
            Execute           := TRUE);

    IF _fbReset.Error
    THEN
      _nErrorId               := _fbReset.ErrorID;
      _eState                 := E_PROGRESS.PROGRESS_ERROR;

      _stMsg.eType            := E_MessageType.eMessageError;
      _stMsg.eSubdevice       := e_Subdevice.fbReset;
      _stMsg.iErrorNumber     := _nErrorId;
      _stMsg.sText            := TO_STRING(_eState);
      f_MessageSet(_stMsg);

    ELSIF NOT _Mover.Status.Moving
    THEN
      _eState                 := E_PROGRESS.PROGRESS_DONE;

      IF (_eMessageLevel > E_MessageType.eMessageError)
      THEN
        _stMsg.eType          := E_MessageType.eMessageInfo;
        _stMsg.eSubdevice     := e_Subdevice.fbReset;
        _stMsg.iErrorNumber   := _nErrorId;
        _stMsg.sText          := TO_STRING(_eState);
        f_MessageSet(_stMsg);
      END_IF
    END_IF
END_CASE
//-----------------------------------------------------------------------------
//-----------------------------------------------------------------------------
CASE _eState
OF
  E_PROGRESS.PROGRESS_ERROR,
  E_PROGRESS.PROGRESS_DONE:
    _stInfo.nErrorId          := _nErrorId;

    _stInfo.bMoverError       :=
	  _bError                   := FALSE;

    _fbReset(
            Axis              := _Mover, 
            Execute           := FALSE);
			
		
END_CASE
//-----------------------------------------------------------------------------
//-----------------------------------------------------------------------------

Reset                         := _eState;
END_METHOD

METHOD SendToAbsPosCa : E_PROGRESS
VAR_INPUT
  Execute             : BOOL;
  stMoveData          : ST_MOVE_DATA;
END_VAR
VAR_INST
  _nErrorId           : UDINT;
  _rPos               : LREAL;
  _rStart             : LREAL;
  _eState             : E_PROGRESS;
END_VAR
IF NOT Execute THEN _eState  := E_PROGRESS.PROGRESS_INIT; END_IF 
IF NOT Check() THEN SendToAbsPosCa   := E_PROGRESS.PROGRESS_ERROR; RETURN; END_IF


CASE _eState
OF
  E_PROGRESS.PROGRESS_INIT:
    IF Execute
    THEN
      _nErrorId               := 0;
      _rStart                 := _Mover.NcToPlc.SetPos;

      _eState                 := E_PROGRESS.PROGRESS_BUSY;
    END_IF
END_CASE
//-----------------------------------------------------------------------------
//-----------------------------------------------------------------------------
CASE _eState
OF
  E_PROGRESS.PROGRESS_BUSY:
    _eState                   := E_PROGRESS.PROGRESS_PREPARE;
    _fbPower.Override         := stMoveData.rOverride;

    _rPos                     := stMoveData.rPos;
	
    _rLastPosition            := _rPos;
    _rLastGap                 := stMoveData.rGap;

    _fbSendAbsCa( 
            Axis              := _Mover, 
            Execute           := FALSE, 
            ContinuousUpdate  := TRUE, 
            Position          := _rPos,
            Velocity          := stMoveData.rVelo, 
            Acceleration      := stMoveData.rAcc, 
            Deceleration      := stMoveData.rAcc, 
            Jerk              := stMoveData.rJerk, 
            Gap               := stMoveData.rGap, 
            BufferMode        := Tc3_Mc3Definitions.MC_BUFFER_MODE.mcAborting);

    IF (_eMessageLevel > E_MessageType.eMessageVerbose)
    THEN
      _stMsg.eType            := E_MessageType.eMessageSentient;
      _stMsg.eSubdevice       := e_Subdevice.fbSendToAbsPosCa;
      _stMsg.iErrorNumber     := _nErrorId;
      _stMsg.sText            := concat(TO_STRING(_eState), ': ');
      _stMsg.sText            := concat(_stMsg.sText, 'stMoveData.rPos: ');
      _stMsg.sText            := concat(_stMsg.sText, TO_STRING(stMoveData.rPos));
      f_MessageSet(_stMsg);

      _stMsg.eType            := E_MessageType.eMessageSentient;
      _stMsg.eSubdevice       := e_Subdevice.fbSendToAbsPosCa;
      _stMsg.iErrorNumber     := _nErrorId;
      _stMsg.sText            := concat(TO_STRING(_eState), ': ');
      _stMsg.sText            := concat(_stMsg.sText, '.rDistance: ');
      _stMsg.sText            := concat(_stMsg.sText, TO_STRING(stMoveData.rDistance));
      f_MessageSet(_stMsg);
    END_IF
END_CASE
//-----------------------------------------------------------------------------
//-----------------------------------------------------------------------------
CASE _eState
OF
  E_PROGRESS.PROGRESS_PREPARE:
    _fbSendAbsCa( 
            Axis              := _Mover, 
            Execute           := TRUE, 
            ContinuousUpdate  := TRUE, 
            Position          := _rPos,
            Velocity          := stMoveData.rVelo, 
            Acceleration      := stMoveData.rAcc, 
            Deceleration      := stMoveData.rAcc, 
            Jerk              := stMoveData.rJerk, 
            Gap               := stMoveData.rGap, 
            BufferMode        := Tc3_Mc3Definitions.MC_BUFFER_MODE.mcAborting);

    IF _fbSendAbsCa.Error
    THEN
      _bError                 := TRUE;
      _nErrorId               := _fbSendAbsCa.ErrorId;
      _stInfo.nErrorId        := _nErrorId;
      _eState                 := E_PROGRESS.PROGRESS_ERROR;

      _stMsg.eType            := E_MessageType.eMessageError;
      _stMsg.eSubdevice       := e_Subdevice.fbSendToAbsPosCa;
      _stMsg.iErrorNumber     := _nErrorId;
      _stMsg.sText            := TO_STRING(_eState);
      f_MessageSet(_stMsg);

    ELSIF _fbSendAbsCa.Active OR
          _fbSendAbsCa.Done
    THEN
      _eState                 := E_PROGRESS.PROGRESS_WORKING;

      IF (_eMessageLevel > E_MessageType.eMessageVerbose)
      THEN
        _stMsg.eType          := E_MessageType.eMessageSentient;
        _stMsg.eSubdevice     := e_Subdevice.fbSendToAbsPosCa;
        _stMsg.iErrorNumber   := _nErrorId;
        _stMsg.sText          := concat(TO_STRING(_eState), ': ');
        _stMsg.sText          := concat(_stMsg.sText, '.SetPos: ');
        _stMsg.sText          := concat(_stMsg.sText, TO_STRING(_Mover.NcToPlc.SetPos));
        //f_MessageSet(_stMsg);
      END_IF
    END_IF
END_CASE
//-----------------------------------------------------------------------------
//-----------------------------------------------------------------------------
CASE _eState
OF
  E_PROGRESS.PROGRESS_WORKING:
    _fbSendAbsCa(
            Axis              := _Mover);

    IF _fbSendAbsCa.Error
    THEN
      _bError                 := TRUE;
      _nErrorId               := _fbSendAbsCa.ErrorId;
      _stInfo.nErrorId        := _nErrorId;
      _fbMoveAbsCa( 
            Axis              := _Mover, 
            Execute           := FALSE);

      _eState                 := E_PROGRESS.PROGRESS_ERROR;

      _stMsg.eType            := E_MessageType.eMessageError;
      _stMsg.eSubdevice       := e_Subdevice.fbSendToAbsPosCa;
      _stMsg.iErrorNumber     := _nErrorId;
      _stMsg.sText            := TO_STRING(_eState);
      f_MessageSet(_stMsg);

    ELSIF (_Mover.NcToPlc.SetPos > _rStart + stMoveData.rDistance)
    THEN
      _eState                 := E_PROGRESS.PROGRESS_DONE;

      IF (_eMessageLevel > E_MessageType.eMessageError)
      THEN
        _stMsg.eType          := E_MessageType.eMessageInfo;
        _stMsg.eSubdevice     := e_Subdevice.fbSendToAbsPosCa;
        _stMsg.iErrorNumber   := _nErrorId;
        _stMsg.sText          := concat(TO_STRING(_eState), ': ');
        _stMsg.sText          := concat(_stMsg.sText, '.SetPos: ');
        _stMsg.sText          := concat(_stMsg.sText, TO_STRING(_Mover.NcToPlc.SetPos));
        _stMsg.sText          := concat(_stMsg.sText, ' ');
        _stMsg.sText          := concat(_stMsg.sText, '.ActVelo: ');
        _stMsg.sText          := concat(_stMsg.sText, TO_STRING(_Mover.NcToPlc.ActVelo));

        f_MessageSet(_stMsg);
      END_IF
      _fbSendAbsCa( 
            Axis              := _Mover, 
            Execute           := FALSE);
    END_IF
END_CASE
//-----------------------------------------------------------------------------
//-----------------------------------------------------------------------------

SendToAbsPosCa                := _eState;
END_METHOD

METHOD SendToModuloPosCa : E_PROGRESS
VAR_INPUT
  Execute             : BOOL;
  stMoveData          : ST_MOVE_DATA;
END_VAR
VAR_INST
  _nErrorId           : UDINT;
  _rPos               : LREAL;
  _rStart             : LREAL;
  _eState             : E_PROGRESS;

  _rModActPos         : lreal;
END_VAR
IF NOT Execute THEN _eState  := E_PROGRESS.PROGRESS_INIT; END_IF 
IF NOT Check() THEN SendToModuloPosCa   := E_PROGRESS.PROGRESS_ERROR; RETURN; END_IF


CASE _eState
OF
  E_PROGRESS.PROGRESS_INIT:
    IF Execute
    THEN
      _nErrorId               := 0;
      _rStart                 := _Mover.NcToPlc.SetPos;

      _eState                 := E_PROGRESS.PROGRESS_BUSY;
    END_IF
    _fbSendAbsCa( 
            Axis              := _Mover, 
            Execute           := FALSE);
END_CASE
//-----------------------------------------------------------------------------
//-----------------------------------------------------------------------------
CASE _eState
OF
  E_PROGRESS.PROGRESS_BUSY:
    _eState                   := E_PROGRESS.PROGRESS_PREPARE;
    _fbPower.Override         := stMoveData.rOverride;

    _rPos                     := ABS(_Mover.NcToPlc.ModuloActTurns)* _RailLength + stMoveData.rPos;
	
    _rLastPosition            := _rPos;
    _rLastGap                 := stMoveData.rGap;

    _fbSendAbsCa( 
            Axis              := _Mover, 
            Execute           := FALSE, 
            ContinuousUpdate  := TRUE, 
            Position          := _rPos,
            Velocity          := stMoveData.rVelo, 
            Acceleration      := stMoveData.rAcc, 
            Deceleration      := stMoveData.rAcc, 
            Jerk              := stMoveData.rJerk, 
            Gap               := stMoveData.rGap, 
            BufferMode        := Tc3_Mc3Definitions.MC_BUFFER_MODE.mcAborting);

    IF (_eMessageLevel > E_MessageType.eMessageVerbose)
    THEN
      _stMsg.eType            := E_MessageType.eMessageSentient;
      _stMsg.eSubdevice       := e_Subdevice.fbSendToModuloPosCa;
      _stMsg.iErrorNumber     := _nErrorId;
      _stMsg.sText            := concat(TO_STRING(_eState), ': ');
      _stMsg.sText            := concat(_stMsg.sText, 'stMoveData.rPos: ');
      _stMsg.sText            := concat(_stMsg.sText, TO_STRING(stMoveData.rPos));
      f_MessageSet(_stMsg);

      _stMsg.eType            := E_MessageType.eMessageSentient;
      _stMsg.eSubdevice       := e_Subdevice.fbSendToModuloPosCa;
      _stMsg.iErrorNumber     := _nErrorId;
      _stMsg.sText            := concat(TO_STRING(_eState), ': ');
      _stMsg.sText            := concat(_stMsg.sText, '.rDistance: ');
      _stMsg.sText            := concat(_stMsg.sText, TO_STRING(stMoveData.rDistance));
      f_MessageSet(_stMsg);

    END_IF
END_CASE
//-----------------------------------------------------------------------------
//-----------------------------------------------------------------------------
CASE _eState
OF
  E_PROGRESS.PROGRESS_PREPARE:
    _fbSendAbsCa( 
            Axis              := _Mover, 
            Execute           := TRUE, 
            ContinuousUpdate  := TRUE, 
            Position          := _rPos,
            Velocity          := stMoveData.rVelo, 
            Acceleration      := stMoveData.rAcc, 
            Deceleration      := stMoveData.rAcc, 
            Jerk              := stMoveData.rJerk, 
            Gap               := stMoveData.rGap, 
            BufferMode        := Tc3_Mc3Definitions.MC_BUFFER_MODE.mcAborting);

    IF _fbSendAbsCa.Error
    THEN
      _bError                 := TRUE;
      _nErrorId               := _fbSendAbsCa.ErrorId;
      _stInfo.nErrorId        := _nErrorId;
      _eState                 := E_PROGRESS.PROGRESS_ERROR;

      _stMsg.eType            := E_MessageType.eMessageError;
      _stMsg.eSubdevice       := e_Subdevice.fbSendToModuloPosCa;
      _stMsg.iErrorNumber     := _nErrorId;
      _stMsg.sText            := TO_STRING(_eState);
      f_MessageSet(_stMsg);

      _fbSendAbsCa( 
            Axis              := _Mover, 
            Execute           := FALSE);

    ELSIF _fbSendAbsCa.Active OR
          _fbSendAbsCa.Done
    THEN
      _eState                 := E_PROGRESS.PROGRESS_WORKING;
      _rModActPos             := Tc2_Math.LMOD(_Mover.NcToPlc.SetPos, _RailLength);

      IF (_eMessageLevel > E_MessageType.eMessageVerbose)
      THEN
        _stMsg.eType          := E_MessageType.eMessageSentient;
        _stMsg.eSubdevice     := e_Subdevice.fbSendToModuloPosCa;
        _stMsg.iErrorNumber   := _nErrorId;
        _stMsg.sText            := concat(TO_STRING(_eState), ': ');
        _stMsg.sText          := concat(_stMsg.sText, '_rModActPos: ');
        _stMsg.sText          := concat(_stMsg.sText, TO_STRING(_rModActPos));
        //f_MessageSet(_stMsg);
      END_IF
(*
    ELSIF (_Mover.NcToPlc.ActPos > _rStart + stMoveData.rDistance)
    THEN
      _eState                 := E_PROGRESS.PROGRESS_DONE;

      IF (_eMessageLevel < E_MessageType.eMessageError)
      THEN
        _stMsg.eType          := E_MessageType.eMessageInfo;
        _stMsg.eSubdevice     := e_Subdevice.fbSendToModuloPosCa;
        _stMsg.iErrorNumber   := _nErrorId;
        _stMsg.sText          := TO_STRING(_eState);
        f_MessageSet(_stMsg);
      END_IF
      _fbMoveAbsCa( 
            Axis              := _Mover, 
            Execute           := FALSE);
*)
    END_IF
END_CASE
//-----------------------------------------------------------------------------
//-----------------------------------------------------------------------------
CASE _eState
OF
  E_PROGRESS.PROGRESS_WORKING:
    _fbSendAbsCa(
            Axis              := _Mover);

    IF _fbSendAbsCa.Error
    THEN
      _bError                 := TRUE;
      _nErrorId               := _fbMoveAbsCa.ErrorId;
      _stInfo.nErrorId        := _nErrorId;
      _fbMoveAbsCa( 
            Axis              := _Mover, 
            Execute           := FALSE);

      _eState                 := E_PROGRESS.PROGRESS_ERROR;

      _stMsg.eType            := E_MessageType.eMessageError;
      _stMsg.eSubdevice       := e_Subdevice.fbSendToModuloPosCa;
      _stMsg.iErrorNumber     := _nErrorId;
      _stMsg.sText            := TO_STRING(_eState);
      f_MessageSet(_stMsg);

    ELSIF (_Mover.NcToPlc.SetPos > _rStart + stMoveData.rDistance)
    THEN
      _eState                 := E_PROGRESS.PROGRESS_DONE;
      _rModActPos             := Tc2_Math.LMOD(_Mover.NcToPlc.SetPos, _RailLength);


      IF (_eMessageLevel > E_MessageType.eMessageError)
      THEN
        _stMsg.eType          := E_MessageType.eMessageInfo;
        _stMsg.eSubdevice     := e_Subdevice.fbSendToModuloPosCa;
        _stMsg.iErrorNumber   := _nErrorId;
        _stMsg.sText          := concat(TO_STRING(_eState), ': ');
        _stMsg.sText          := concat(_stMsg.sText, '_rModActPos: ');
        _stMsg.sText          := concat(_stMsg.sText, TO_STRING(_rModActPos));
        _stMsg.sText          := concat(_stMsg.sText, ' ');
        _stMsg.sText          := concat(_stMsg.sText, '.ActVelo: ');
        _stMsg.sText          := concat(_stMsg.sText, TO_STRING(_Mover.NcToPlc.ActVelo));
        f_MessageSet(_stMsg);
      END_IF
      _fbSendAbsCa( 
            Axis              := _Mover, 
            Execute           := FALSE);
    END_IF
END_CASE
//-----------------------------------------------------------------------------
//-----------------------------------------------------------------------------

SendToModuloPosCa                   := _eState;
END_METHOD

METHOD Stop : E_PROGRESS
VAR_INPUT
  Execute             : BOOL;
  stMoveData          : ST_MOVE_DATA;
END_VAR
VAR_INST
  _nErrorId           : UDINT;
  _eState             : E_PROGRESS;
END_VAR
IF NOT Execute 
THEN 
	_eState := E_PROGRESS.PROGRESS_INIT; 
END_IF 
IF NOT Check() 
THEN 
	Stop := E_PROGRESS.PROGRESS_ERROR; 
	RETURN; 
END_IF


CASE _eState
OF
  E_PROGRESS.PROGRESS_INIT:
    IF Execute
    THEN
      _nErrorId               := 0;
      _eState                 := E_PROGRESS.PROGRESS_BUSY;
    END_IF
END_CASE
//-----------------------------------------------------------------------------
//-----------------------------------------------------------------------------
CASE _eState
OF
  E_PROGRESS.PROGRESS_BUSY:
    _eState                   := E_PROGRESS.PROGRESS_PREPARE;
    _fbStop(
            Axis              := _Mover, 
            Execute           := FALSE, 
            Deceleration      := stMoveData.rAcc, 
            Jerk              := stMoveData.rJerk); 

    IF (_eMessageLevel > E_MessageType.eMessageInfo)
    THEN
      _stMsg.eType            := E_MessageType.eMessageVerbose;
      _stMsg.eSubdevice       := e_Subdevice.fbStop;
      _stMsg.iErrorNumber     := _nErrorId;
      _stMsg.sText            := TO_STRING(_eState);
      f_MessageSet(_stMsg);
    END_IF
END_CASE
//-----------------------------------------------------------------------------
//-----------------------------------------------------------------------------
CASE _eState
OF
  E_PROGRESS.PROGRESS_PREPARE:
    _fbStop(Axis              := _Mover, 
            Execute           := TRUE, 
            Deceleration      := stMoveData.rAcc, 
            Jerk              := stMoveData.rJerk);

    IF _fbStop.Error
    THEN
      _bError                 := TRUE;
      _nErrorId               := _fbStop.ErrorID;
      _eState                 := E_PROGRESS.PROGRESS_ERROR;

      _stMsg.eType            := E_MessageType.eMessageError;
      _stMsg.eSubdevice       := e_Subdevice.fbStop;
      _stMsg.iErrorNumber     := _nErrorId;
      _stMsg.sText            := TO_STRING(_eState);
      f_MessageSet(_stMsg);

    ELSIF _fbStop.Done
    THEN
      _eState                 := E_PROGRESS.PROGRESS_DONE;

      IF (_eMessageLevel > E_MessageType.eMessageError)
      THEN
        _stMsg.eType          := E_MessageType.eMessageInfo;
        _stMsg.eSubdevice     := e_Subdevice.fbStop;
        _stMsg.iErrorNumber   := _nErrorId;
        _stMsg.sText          := TO_STRING(_eState);
        f_MessageSet(_stMsg);
      END_IF
    END_IF
END_CASE
//-----------------------------------------------------------------------------
//-----------------------------------------------------------------------------
CASE _eState
OF
  E_PROGRESS.PROGRESS_ERROR,
  E_PROGRESS.PROGRESS_DONE:
    _stInfo.nErrorId          := _nErrorId;
    _fbStop(
            Axis              := _Mover, 
            Execute           := FALSE);
END_CASE
//-----------------------------------------------------------------------------
//-----------------------------------------------------------------------------

Stop                          := _eState;
END_METHOD

END_FUNCTION_BLOCK

(* stored: Version 1.1.0.1, ProductVersion 3.1.4026.13
   POU fb_Mover: Id {0329c584-f72c-48ef-81e9-d36f2b915502}, SpecialFunc None
   Folder methods: Id {d4f48e59-bafb-4a6b-a547-9f57a3dde1b3}
   Folder properties: Id {9b756c45-f31b-4fd8-944d-37c13ea518e9}
   Method Check: Id {7aad3024-4d91-4070-bd1c-7ab21c07b418}
   Method Cycle: Id {23c9e7eb-0f59-4742-a92e-59fc57018459}
   Method Disable: Id {097d7d29-677b-4897-9517-c610ca359790}
   Method Enable: Id {5c42fddf-2f46-4658-9cfe-4e104b612772}
   Method GearIn: Id {eb68f991-484a-4638-a27c-6c851ba6b822}
   Method GearInPosCa: Id {1420a175-40e0-489e-92fe-2ab56883c746}
   Method GearOut: Id {6d9377d6-ed75-428d-ab8c-7faa8f3f3051}
   Method Halt: Id {6d1913d1-ebf7-491a-a13e-d4ef262d26ef}
   Method HaltCa: Id {1df8e06f-9c25-47b7-a0ee-0f8e224033c8}
   Property LastGap: Id {b5ed76e9-676f-4353-b13a-0502ca2acc9a}
   Set Set: Id {f4acb2e9-9d40-45c9-a29c-1e724dd24870}
   Property LastPosition: Id {bfd53c64-02d7-4b58-bd3b-f27b62fcf723}
   Set Set: Id {eec85df7-ac46-4292-9d60-1e007a9091f1}
   Property Master: Id {b6e3b62d-f089-480e-82df-cbd05240e555}
   Set Set: Id {b16aaec0-0d1a-4ab3-bb6b-8afa2d833253}
   Property MessageLevel: Id {a0a14a73-1391-4431-9bc4-6a06d816fc4c}
   Set Set: Id {61cac132-b30e-4323-bc53-0173e0abd77d}
   Property ModuloTurn: Id {29a92467-8779-409e-8918-3e94f26a126b}
   Get Get: Id {abdb873d-00f6-4125-8476-07cb84d6957b}
   Property Mover: Id {725f2a78-1f2c-4af9-8ce5-bb55abd5bdc7}
   Set Set: Id {f63f36af-a1b3-44d0-911f-8078223fe58a}
   Property MoverId: Id {0ba03e0e-28d1-4142-b9f5-7e4ec07c6988}
   Set Set: Id {c36f4173-a354-4b08-9d63-481abb7f409a}
   Property MoverInfo: Id {37db38a4-3c3d-40a1-a24e-7c3e5a8f6c0d}
   Set Set: Id {09a628eb-fb2a-4de3-b247-fb2dd797a92f}
   Method MoveToPos: Id {fb779f0f-ad18-4dac-8c8b-6a09fac8cfc2}
   Method MoveToPosCa: Id {d4a8c4a1-971b-4d94-815f-d0a216b18ca8}
   Property RailLength: Id {d97d4601-f98a-4fd6-a9df-28f8fa09e071}
   Get Get: Id {8260a61c-9381-468f-9345-10dfc6582380}
   Set Set: Id {2d590b04-104f-41d4-b68a-2a40bc95b2e9}
   Method Reset: Id {f267dfd0-7a70-4720-839c-88e90bbf285e}
   Method SendToAbsPosCa: Id {d7ea3c10-bae0-4cbd-97d2-8fcc9da3c276}
   Method SendToModuloPosCa: Id {42c54723-2fdd-42ff-a93c-927000ec8f99}
   Method Stop: Id {791a388a-a298-41ba-80ec-d761701c9846} *)
